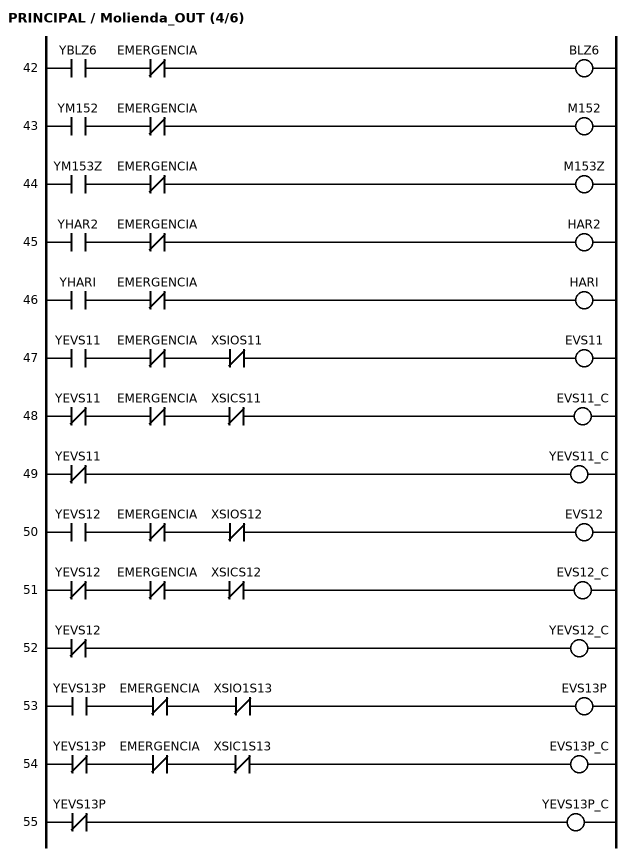
; [picture p72: PRINCIPAL / Molienda_OUT, rungs 42-55]
; rung 42
LD YBLZ6
ANDNOT EMERGENCIA
OUT BLZ6
; rung 43
LD YM152
ANDNOT EMERGENCIA
OUT M152
; rung 44
LD YM153Z
ANDNOT EMERGENCIA
OUT M153Z
; rung 45
LD YHAR2
ANDNOT EMERGENCIA
OUT HAR2
; rung 46
LD YHARI
ANDNOT EMERGENCIA
OUT HARI
; rung 47
LD YEVS11
ANDNOT EMERGENCIA
ANDNOT XSIOS11
OUT EVS11
; rung 48
LDNOT YEVS11
ANDNOT EMERGENCIA
ANDNOT XSICS11
OUT EVS11_C
; rung 49
LDNOT YEVS11
OUT YEVS11_C
; rung 50
LD YEVS12
ANDNOT EMERGENCIA
ANDNOT XSIOS12
OUT EVS12
; rung 51
LDNOT YEVS12
ANDNOT EMERGENCIA
ANDNOT XSICS12
OUT EVS12_C
; rung 52
LDNOT YEVS12
OUT YEVS12_C
; rung 53
LD YEVS13P
ANDNOT EMERGENCIA
ANDNOT XSIO1S13
OUT EVS13P
; rung 54
LDNOT YEVS13P
ANDNOT EMERGENCIA
ANDNOT XSIC1S13
OUT EVS13P_C
; rung 55
LDNOT YEVS13P
OUT YEVS13P_C

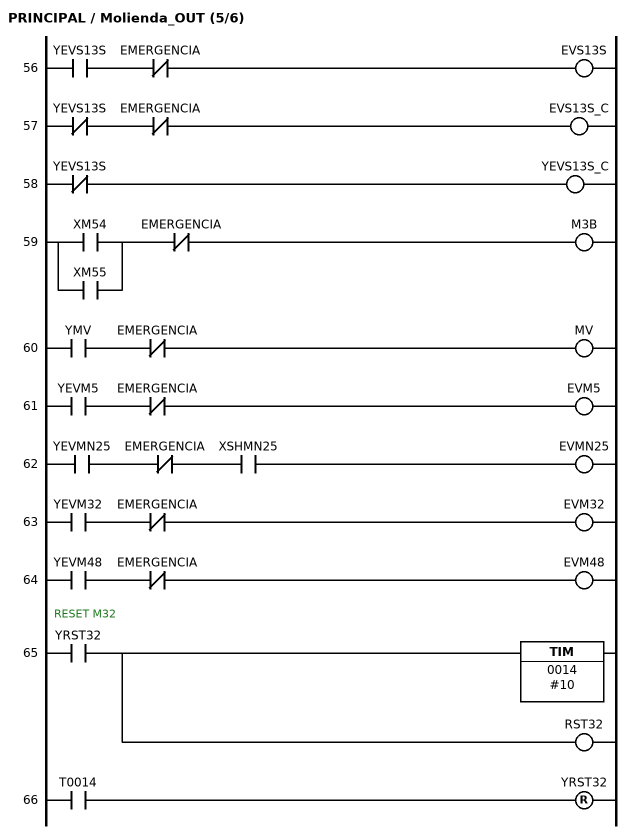
; rung 56
LD YEVS13S
ANDNOT EMERGENCIA
OUT EVS13S
; rung 57
LDNOT YEVS13S
ANDNOT EMERGENCIA
OUT EVS13S_C
; rung 58
LDNOT YEVS13S
OUT YEVS13S_C
; rung 59
LD XM54
OR XM55
ANDNOT EMERGENCIA
OUT M3B
; rung 60
LD YMV
ANDNOT EMERGENCIA
OUT MV
; rung 61
LD YEVM5
ANDNOT EMERGENCIA
OUT EVM5
; rung 62
LD YEVMN25
ANDNOT EMERGENCIA
AND XSHMN25
OUT EVMN25
; rung 63
LD YEVM32
ANDNOT EMERGENCIA
OUT EVM32
; rung 64
LD YEVM48
ANDNOT EMERGENCIA
OUT EVM48
; rung 65: RESET M32
LD YRST32
TIM 0014 #10
OUT RST32
; rung 66
LD T0014
RSET YRST32

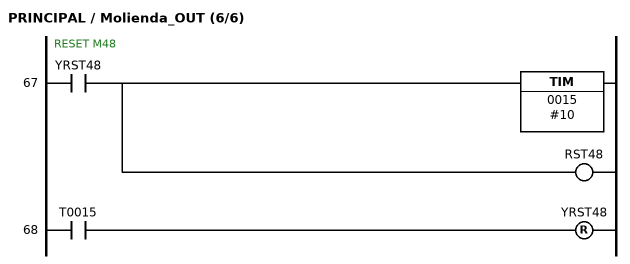
; rung 67: RESET M48
LD YRST48
TIM 0015 #10
OUT RST48
; rung 68
LD T0015
RSET YRST48

### Section FIN
; rung 0
END(001)